FUNCTION GetDistanceToPositionFromBase2D : LREAL
VAR_INPUT
	position : Position;	//The target position
END_VAR
VAR
	xSide : LREAL;
	zSide : LREAL;
END_VAR

xSide := GetXSide(position.x);
zSide := GetZSide(position.z);

GetDistanceToPositionFromBase2D := GetHypotenuse(xSide, zSide);

END_FUNCTION

(* stored: Version 1.1.0.1, ProductVersion 3.1.4024.12
   POU GetDistanceToPositionFromBase2D: Id {33e46975-d7ec-4981-bcfc-0cffb29d096e}, SpecialFunc None *)
